TYPE ST_PowerControl_Events :
STRUCT
	b_ReactivePIDError			: BOOL;
	b_ActivePIDError			: BOOL;
	b_FreqShiftPIDError			: BOOL;
END_STRUCT
END_TYPE

(* stored: Version 1.1.0.1, ProductVersion 3.1.4026.18
   DUT ST_PowerControl_Events: Id {dcb98ebd-43b8-40a7-a23e-d5ccf30658ed} *)
